{attribute 'GeneratedUsingTerminal: AES-D-BC-ECAT-0000'}
{attribute addProperty BoxType "AES-D-BC-ECAT-0000"}
{attribute addProperty Id "digital_Data_IAT %I*ARRAY[0..27] OF USINT28"}
{attribute addProperty CRC "2446583242"}
{attribute addProperty Size "28"}
TYPE Inputs_03C60166 EXTENDS TcoIo.InputBase_8311D824 :
STRUCT
	{attribute addProperty Name "digital_Data_I"}
	digital_Data_I AT %I* : ARRAY[0..27] OF USINT;
END_STRUCT
END_TYPE

(* stored: Version 1.2.0.0, ProductVersion 3.1.4024.11
   DUT Inputs_03C60166: Id {a0201f89-3104-0eac-3a56-fa75b0ca6016} *)
